(* PLC project Tc2_Utilities.FB_CSVMemBufferWriter Demo, tc3-libraries-kb TwinCAT 3.1 *)
(* stored: creationDateTime 2026-05-10T20:00:00, modificationDateTime 2026-05-10T20:00:00 *)

PROGRAM P_Demo_FB_CSVMemBufferWriter
  VAR
    fbFB_CSVMemBufferWriter : FB_CSVMemBufferWriter;  (* Tc2_Utilities.FB_CSVMemBufferWriter 实例 *)
    arg_eCmd : E_EnumCmdType;  (* VAR_INPUT eCmd *)
    arg_putValue : T_MaxString;  (* VAR_INPUT putValue *)
    arg_pValue : POINTER TO BYTE;  (* VAR_INPUT pValue *)
    arg_cbValue : UDINT;  (* VAR_INPUT cbValue *)
    arg_bCRLF : BOOL;  (* VAR_INPUT bCRLF *)
    arg_pBuffer : POINTER TO BYTE;  (* VAR_INPUT pBuffer *)
    arg_cbBuffer : UDINT;  (* VAR_INPUT cbBuffer *)
    out_bOk : BOOL;  (* VAR_OUTPUT bOk *)
    out_cbSize : UDINT;  (* VAR_OUTPUT cbSize *)
    out_cbFree : UDINT;  (* VAR_OUTPUT cbFree *)
    out_nFields : UDINT;  (* VAR_OUTPUT nFields *)
    out_nRecords : UDINT;  (* VAR_OUTPUT nRecords *)
    out_cbWrite : UDINT;  (* VAR_OUTPUT cbWrite *)
  END_VAR

            // ============================================================
// Tc2_Utilities.FB_CSVMemBufferWriter 演示程序（FB 实例）
// ============================================================
// 验证步骤：
//   1. 引用 Tc2_Utilities（及依赖类型所在库 Tc2_System 等）
//   2. 编译 + 登录
//   3. 按 doc.md 给 arg_* 赋值
//   4. 在线监视 out_* / io_* 输出
// ============================================================

fbFB_CSVMemBufferWriter(
    eCmd := arg_eCmd,
    putValue := arg_putValue,
    pValue := arg_pValue,
    cbValue := arg_cbValue,
    bCRLF := arg_bCRLF,
    pBuffer := arg_pBuffer,
    cbBuffer := arg_cbBuffer,
    bOk => out_bOk,
    cbSize => out_cbSize,
    cbFree => out_cbFree,
    nFields => out_nFields,
    nRecords => out_nRecords,
    cbWrite => out_cbWrite
);

          
END_PROGRAM
